{attribute 'qualified_only'}
{attribute 'strict'}
TYPE E_Axis :
(
	TakeY:=1,
	TakeZ,
	UC_Y
);
END_TYPE

(* stored: Version 1.1.0.1, ProductVersion 3.1.4024.3
   DUT E_Axis: Id {dea5fc20-99f0-44fb-afc9-fcc770b9d710} *)
